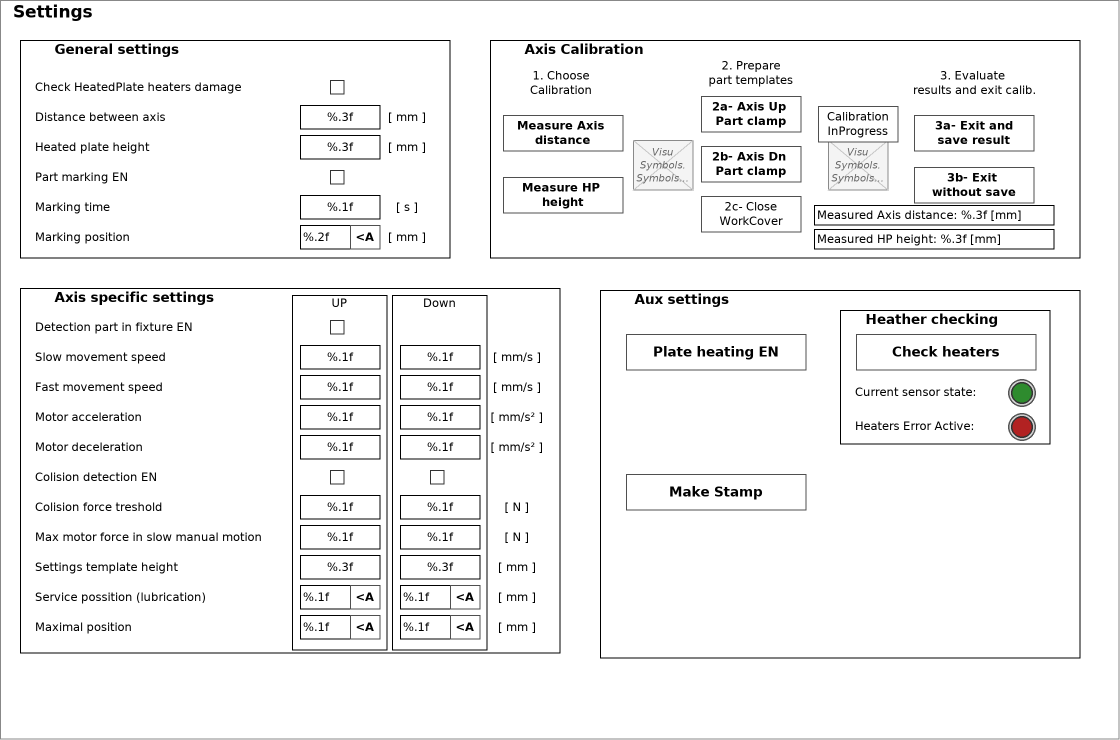
VISUALIZATION vHP3_MachineSub_Settings  // 1120x740
VAR_IN_OUT
	fbHP: fbHPv3_Control;
END_VAR
    RoundedRectangle (20,288 540x365), "Axis specific settings"
    RoundedRectangle (392,295 95x355), "Down"
    RoundedRectangle (292,295 95x355), "UP"
    RoundedRectangle (20,40 430x218), "General settings"
    RoundedRectangle (490,40 590x218), "Axis Calibration"
    Label (32,75 260x24), "Check HeatedPlate heaters damage"
    Label (32,105 260x24), "Distance between axis"
    Rectangle (300,105 80x24), "%.3f", text variable: fbHP.stMachSettings.lrAxisDIstance_mm
        OnMouseDown: write the text variable via Default, min 0.1, max 5, title 'Test drawer time', format %.1f
    Label (382,105 50x24), "[ mm ]"
    Checkbox (328,75 24x24), variable: fbHP.stMachSettings.bCheckHeatersDamage_EN
    Label (32,135 260x24), "Heated plate height"
    Rectangle (300,135 80x24), "%.3f", text variable: fbHP.stMachSettings.lrHeatedPlateHeight_mm
        OnMouseDown: write the text variable via Default, min 0.1, max 5, title 'Test drawer time', format %.1f
    Label (382,135 50x24), "[ mm ]"
    Label (32,165 260x24), "Part marking EN"
    Checkbox (328,165 24x24), variable: fbHP.stMachSettings.bPartMarking_EN, input disabled if: NOT fbHP.bMarkingAsembled
    Label (32,195 260x24), "Marking time"
    Rectangle (300,195 80x24), "%.1f", text variable: fbHP.stMachSettings.rPartMarkingTime, input disabled if: NOT fbHP.bMarkingAsembled
        OnMouseDown: write the text variable via Default, min 0.1, max 5, title 'Test drawer time', format %.1f
    Label (382,195 50x24), "[ s ]"
    Label (32,405 260x24), "Motor acceleration"
    Rectangle (300,405 80x24), "%.1f", text variable: fbHP.stMachSettings.stAxisUpSettings.rAcceleration
        OnMouseDown: write the text variable via Default, min 100, max 5000, title 'Acceleration', format %.1f
    Label (492,405 50x24), "[ mm/s² ]"
    Label (32,435 260x24), "Motor deceleration"
    Rectangle (300,435 80x24), "%.1f", text variable: fbHP.stMachSettings.stAxisUpSettings.rDeceleration
        OnMouseDown: write the text variable via Default, min 100, max 5000, title 'Deceleration', format %.1f
    Label (492,435 50x24), "[ mm/s² ]"
    Label (32,555 260x24), "Settings template height"
    Rectangle (300,555 80x24), "%.3f", text variable: fbHP.stMachSettings.stAxisUpSettings.lrSettingTemplateHeight_mm
        OnMouseDown: write the text variable via Default, min 10, max 300, title 'Setting template height', format %.1f
    Label (492,555 50x24), "[ mm ]"
    Label (32,585 260x24), "Service possition (lubrication)"
    Rectangle (300,585 80x24), "%.1f", text variable: fbHP.stMachSettings.stAxisUpSettings.lrService_Pos_mm
        OnMouseDown: write the text variable via Default, min 0, max 300, title 'Service position', format %.1f
    Label (492,585 50x24), "[ mm ]"
    Label (32,615 260x24), "Maximal position"
    Rectangle (300,615 80x24), "%.1f", text variable: fbHP.stMachSettings.stAxisUpSettings.lrMax_Pos
        OnMouseDown: write the text variable via Default, min 100, max 300, title 'Max possition', format %.1f
    Label (492,615 50x24), "[ mm ]"
    Label (32,225 260x24), "Marking position"
    Label (382,225 50x24), "[ mm ]"
    Rectangle (400,405 80x24), "%.1f", text variable: fbHP.stMachSettings.stAxisDnSettings.rAcceleration
        OnMouseDown: write the text variable via Default, min 100, max 5000, title 'Acceleration', format %.1f
    Rectangle (400,435 80x24), "%.1f", text variable: fbHP.stMachSettings.stAxisDnSettings.rDeceleration
        OnMouseDown: write the text variable via Default, min 100, max 5000, title 'Deceleration', format %.1f
    Rectangle (400,555 80x24), "%.3f", text variable: fbHP.stMachSettings.stAxisDnSettings.lrSettingTemplateHeight_mm
        OnMouseDown: write the text variable via Default, min 10, max 300, title 'Setting template height', format %.1f
    Rectangle (400,585 80x24), "%.1f", text variable: fbHP.stMachSettings.stAxisDnSettings.lrService_Pos_mm
        OnMouseDown: write the text variable via Default, min 0, max 300, title 'Service position', format %.1f
    Rectangle (400,615 80x24), "%.1f", text variable: fbHP.stMachSettings.stAxisDnSettings.lrMax_Pos
        OnMouseDown: write the text variable via Default, min 100, max 300, title 'Max possition', format %.1f
    Rectangle (300,225 80x24), "%.2f", text variable: fbHP.stMachSettings.lrMarking_Pos_mm, input disabled if: NOT fbHP.bMarkingAsembled
        OnMouseDown: write the text variable via Default, min 0, max 200, title 'Marking possition', format %.1f
    Label (32,525 260x24), "Max motor force in slow manual motion"
    Rectangle (300,525 80x24), "%.1f", text variable: fbHP.stMachSettings.stAxisUpSettings.rManualModeMaxForceAtSlow
        OnMouseDown: write the text variable via Default, min 0, max 300, title 'Max force at slow manual move', format %.1f
    Label (492,525 50x24), "[ N ]"
    Rectangle (400,525 80x24), "%.1f", text variable: fbHP.stMachSettings.stAxisDnSettings.rManualModeMaxForceAtSlow
        OnMouseDown: write the text variable via Default, min 0, max 300, title 'Max force at slow manual move', format %.1f
    Label (32,315 260x24), "Detection part in fixture EN"
    Checkbox (328,315 24x24), variable: fbHP.stMachSettings.stAxisUpSettings. bPartInFixtureDetection_EN
    Label (32,345 260x24), "Slow movement speed"
    Rectangle (300,345 80x24), "%.1f", text variable: fbHP.stMachSettings.stAxisUpSettings.rSlowSpeed_mm_s
        OnMouseDown: write the text variable via Default, min 0.5, max 10, title 'Slow speed', format %.1f
    Label (492,345 50x24), "[ mm/s ]"
    Label (32,375 260x24), "Fast movement speed"
    Rectangle (300,375 80x24), "%.1f", text variable: fbHP.stMachSettings.stAxisUpSettings.rFastSpeed_mm_s
        OnMouseDown: write the text variable via Default, min 50, max 320, title 'Fast speed', format %.1f
    Label (492,375 50x24), "[ mm/s ]"
    Rectangle (400,345 80x24), "%.1f", text variable: fbHP.stMachSettings.stAxisDnSettings.rSlowSpeed_mm_s
        OnMouseDown: write the text variable via Default, min 0.5, max 10, title 'Slow speed', format %.1f
    Rectangle (400,375 80x24), "%.1f", text variable: fbHP.stMachSettings.stAxisDnSettings.rFastSpeed_mm_s
        OnMouseDown: write the text variable via Default, min 50, max 320, title 'Fast speed', format %.1f
    Label (32,465 260x24), "Colision detection EN"
    Checkbox (328,465 24x24), variable: fbHP.stMachSettings.stAxisUpSettings.bColisionDettection_EN
    Label (32,495 260x24), "Colision force treshold"
    Rectangle (300,495 80x24), "%.1f", text variable: fbHP.stMachSettings.stAxisUpSettings.rCollisionDetectForce_N
        OnMouseDown: write the text variable via Default, min 2, max 100, title 'Colision detection force', format %.1f
    Label (492,495 50x24), "[ N ]"
    Rectangle (400,495 80x24), "%.1f", text variable: fbHP.stMachSettings.stAxisDnSettings.rCollisionDetectForce_N
        OnMouseDown: write the text variable via Default, min 2, max 100, title 'Colision detection force', format %.1f
    Checkbox (428,465 24x24), variable: fbHP.stMachSettings.stAxisDnSettings.bColisionDettection_EN
    Rectangle (503,115 120x36), "Measure Axis distance", colour toggle: fbHP.bMeasureAxisDistance
        toggle fbHP.bMeasureAxisDistance
    Rectangle (503,177 120x36), "Measure HP height", colour toggle: fbHP.bMeasureHPHeight
        toggle fbHP.bMeasureHPHeight
    Rectangle (914,115 120x36), "3a- Exit and save result", colour toggle: fbHP.iWorkStep = 75, input disabled if: fbHP.iWorkStep <> 75
        toggle fbHP.bHMI_CalibrationSaveResult
    Rectangle (914,167 120x36), "3b- Exit without save", colour toggle: fbHP.iWorkStep = 75, input disabled if: fbHP.iWorkStep <> 75
        toggle fbHP.bHMI_CloseWithoutSaveResult
    Rectangle (701,96 100x36), "2a- Axis Up Part clamp", colour toggle: fbHP.fbAxisUp.PartClamp, input disabled if: (NOT (fbHP.bMeasureAxisDistance OR fbHP.bMeasureHPHeight)) OR fbHP.iWorkStep <> 60
        toggle fbHP.fbAxisUp.stInOuts.bQ_PartLockPiston
    Rectangle (701,146 100x36), "2b- Axis Dn Part clamp", colour toggle: fbHP.fbAxisDn.PartClamp, input disabled if: (NOT (fbHP.bMeasureAxisDistance OR fbHP.bMeasureHPHeight)) OR fbHP.iWorkStep <> 60
        toggle fbHP.fbAxisDn.stInOuts.bQ_PartLockPiston
    Image (633,140 60x50), image: VisuSymbols.Symbols.ArrowBoldRight
    Rectangle (701,196 100x36), "2c- Close WorkCover", colour toggle: fbHP.stInOuts.bI_Sft_WorkCoverClosed, input disabled if: (NOT (fbHP.bMeasureAxisDistance OR fbHP.bMeasureHPHeight)) OR fbHP.iWorkStep <> 60
    Label (501,65 120x36), "1. Choose Calibration"
    Label (701,55 100x36), "2. Prepare part templates"
    Image (828,140 60x50), image: VisuSymbols.Symbols.ArrowBoldRight
    Rectangle (818,106 80x36), "Calibration InProgress", colour toggle: fbHP.iWorkStep > 60 AND fbHP.iWorkStep < 75, input disabled if: NOT (fbHP.bMeasureAxisDistance OR fbHP.bMeasureHPHeight)
    Label (906,65 137x36), "3. Evaluate results and exit calib."
    Rectangle (350,225 30x24), "<A", input disabled if: NOT fbHP.bMarkingAsembled
        OnMouseClick: execute { fbHP.stMachSettings.lrMarking_Pos_mm := fbHP.fbAxisDn.ActualPosition; }
    Rectangle (350,585 30x24), "<A"
        OnMouseClick: execute { fbHP.stMachSettings.stAxisUpSettings.lrService_Pos_mm := fbHP.fbAxisUp.ActualPosition; }
    Rectangle (350,615 30x24), "<A"
        OnMouseClick: execute { fbHP.stMachSettings.stAxisUpSettings.lrMax_Pos := fbHP.fbAxisUp.ActualPosition; }
    Rectangle (450,615 30x24), "<A"
        OnMouseClick: execute { fbHP.stMachSettings.stAxisDnSettings.lrMax_Pos := fbHP.fbAxisDn.ActualPosition; }
    Rectangle (450,585 30x24), "<A"
        OnMouseClick: execute { fbHP.stMachSettings.stAxisDnSettings.lrService_Pos_mm := fbHP.fbAxisDn.ActualPosition; }
    RoundedRectangle (600,290 480x368), "Aux settings"
    Rectangle (626,334 180x36), "Plate heating EN", colour toggle: fbHP.bHeatedPlate_HeatON
        toggle fbHP.bHeatedPlate_HeatON
    RoundedRectangle (10,0 300x26), "Settings"
    Rectangle (626,474 180x36), "Make Stamp", colour toggle: fbHP.bMakeStamp, input disabled if: NOT fbHP.bMarkingAsembled
        toggle fbHP.bMakeStamp
    RoundedRectangle (840,310 210x134), "Heather checking"
    Rectangle (856,334 180x36), "Check heaters", colour toggle: fbHP.iCheckHeaterStep = 10
        toggle fbHP.bExecHeaterCheck
    Lamp1 (1006,377 32x32), variable: fbHP.stInOuts.bI_HeaterCurrentSensor, style: Lamp-Lamp1-Green
    Label (852,380 152x24), "Current sensor state:"
    Label (852,414 152x24), "Heaters Error Active:"
    Lamp1 (1006,411 32x32), variable: fbHP.bHeatersError, style: Lamp-Lamp1-Red
    Rectangle (814,205 240x20), "Measured Axis distance: %.3f [mm]", text variable: fbHP.lrMeasuredAxisDistance, invisible if: NOT fbHP.bMeasureAxisDistance
    Rectangle (814,229 240x20), "Measured HP height: %.3f [mm]", text variable: fbHP.lrMeasuredHPHeight, invisible if: NOT fbHP.bMeasureHPHeight
END_VISUALIZATION

(* stored: Version 1.1.0.1, ProductVersion 3.1.4024.13
   Visu vHP3_MachineSub_Settings: Id {3ece95a6-fc3e-4691-b086-93feb9c630b8} *)
